FUNCTION F_ScrollBarY (* Compute Container_Scrollbar_Content.Top (s16Yposition for Q_ChildPosition) from the current row position: i32BarBaseOffset + (i32Pos * i32BarTravel) / i32PosMax. *)
  (* Standard: 61499-2; Description: Copyright (c) 2026 Meisterschulen am Ostbahnhof This program and the accompanying materials are made available under the terms of the Eclipse Public License 2.0 which is available at https://www.eclipse.org/legal/epl-2.0/ SPDX-License-Identifier: EPL-2.0 *)
  (* Version 1.0, 2026-08-09, Franz Höpfinger, Meisterschulen am Ostbahnhof, initial API and implementation and/or initial documentation *)
  PACKAGE isobus::UT::Q::helpers;
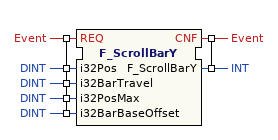
  EVENT_INPUT
    REQ WITH i32Pos, i32BarTravel, i32PosMax, i32BarBaseOffset;
  END_EVENT
  EVENT_OUTPUT
    CNF WITH F_ScrollBarY;
  END_EVENT
  VAR_INPUT
    i32Pos : DINT;
    i32BarTravel : DINT;
    i32PosMax : DINT;
    i32BarBaseOffset : DINT;
  END_VAR
  VAR_OUTPUT
    F_ScrollBarY : INT;
  END_VAR
  BODY IN ST:
PACKAGE isobus::UT::Q::helpers;

(* Compute Container_Scrollbar_Content.Top (s16Yposition for Q_ChildPosition) from the
 * current row position: i32BarBaseOffset + (i32Pos * i32BarTravel) / i32PosMax. *)
FUNCTION F_ScrollBarY : INT

VAR_INPUT
	i32Pos : DINT;
	i32BarTravel : DINT;
	i32PosMax : DINT;
	i32BarBaseOffset : DINT;
END_VAR

F_ScrollBarY := DINT_TO_INT(i32BarBaseOffset + (i32Pos * i32BarTravel) / i32PosMax);

END_FUNCTION
  END_BODY
END_FUNCTION
